// TIA Portal V18 export
TYPE "UDT_Vitotronic100_Params"
// stored: IsFailsafeCompliant false
   STRUCT
      "Actual system output - value" : Array[0..2] of Real;
      "Boiler output value" : Array[0..2] of Real;
      "Burner output" : Array[0..2] of Real;
      "Maximum boiler temperature" : Array[0..2] of Real;
      "Minimum boiler temperature" : Array[0..2] of Real;
      "Set boiler output (effective)" : Array[0..2] of Real;
      "Set boiler water temperature (effective)" : Array[0..2] of Real;
   END_STRUCT;
END_TYPE
